// Core §3.8 — pluggable recipe/type-data source. Implementations MUST validate
// completeness and SchemaVersion before filling ParCfg (migrate-or-fault; never partial).
// Queryable (like I_Module) so a root can ask a provider for I_RecipeStore (§3.8a).
INTERFACE I_RecipeProvider EXTENDS __System.IQueryInterface

// fills the caller's ParCfg; FALSE => caller faults with RECIPE_INVALID (Core §3.8)
METHOD Load : BOOL
VAR_INPUT
    ModelCode : STRING;
    RecipeKey : STRING;
    pParCfg : PVOID;
    Size    : UDINT;
END_VAR
END_METHOD

PROPERTY Ready : BOOL
GET
END_GET
END_PROPERTY

PROPERTY Source : E_RecipeSource
GET
END_GET
END_PROPERTY

END_INTERFACE

(* stored: Version 1.1.0.1, ProductVersion 3.1.4024.12
   Itf I_RecipeProvider: Id {343b29b6-6c9b-4dff-8483-d670a32a9c57}
   Method Load: Id {8fa7419b-404e-4f51-91cd-f16b536e2f37}
   Property Ready: Id {c13e20aa-a9c9-4995-b55d-9b38b7fcf8a4}
   Get Get: Id {cc8a3b6e-ee14-48d3-b6d3-fb4a486f99d6}
   Property Source: Id {16a9a0c3-2e45-4dfa-88da-b93bb02f85c7}
   Get Get: Id {25ff2277-ee7f-412c-8af1-f4670e65513a} *)
